Staubli VAL3: setHome.pgx

public program setHome(num x_nAxisNum, bool& x_bRes)
  local bool l_bError
  local num l_nEtape
  local string l_sMsg
  local num l_nTps
  local bool l_bVerrou
  local bool l_bOK
  local num l_nDuration
  local string l_sYN[2]
  local num l_nDrvPos
begin
  //对绝对编码器电机设置当前值位为零点
    if !isPowered()
      popUpMsg("请先上电")
      return
    endIf
    x_bRes=false
    doStartHoming[x_nAxisNum]=false
    delay(0.1)
    aioSet(aoWorkMode[x_nAxisNum],cst:nHOMINGMODE)
    doStartHoming[x_nAxisNum]=true
    wait(diHomingReached[x_nAxisNum]==false)
    wait(diHomingReached[x_nAxisNum]==true)
    if watch(diHomingReached[x_nAxisNum]==true,2)
      x_bRes=true
      popUpMsg("设置成功")
    endIf
    disablePower()
    delay(0.008)
    aioSet(aoWorkMode[x_nAxisNum],cst:nINTERPMODE)
 end
